PROGRAM MAIN
VAR
	fbSerialCommInstance1 : SerialCom;
	sRecieveString : STRING;
	bRecieveError : BOOL;
	bSendBusy: BOOL;
	eSendError: INT;
	sSendData : STRING;
	bsendTrigger: BOOL;
	STxBuffer: INT;
	tSendTime: INT;
	sizeoff : UINT;
	bRecieveReset: BOOL;
END_VAR

(* Send & Recieve String Data *)
fbSerialCommInstance1(bSendData:= bsendTrigger,
					  bReset := bRecieveReset,
					  TxBuffer := SerialComm.TxBufferPcCom,
					  sSendPrefix:='$01',
					  sSendSuffix:='$02',
					  sSendString:=sSendData,
					  bSendBusy =>bSendBusy,
					  eSendError =>eSendError,
					  RxBuffer := SerialComm.RxBufferPcCom,
					  sReceiveString =>sRecieveString,
					  sReceivePrefix:='$01',
					  sReceiveSuffix:='$02',
					  tReceiveTimeOut := T#1S,
					  bReset :=bRecieveError,
					  bReceiveStringData =>,
					  bReceiveBusy =>,
					  eReceiveError =>,
					  bReceiveTimeOut =>
					  );

END_PROGRAM

(* stored: Version 1.1.0.1, ProductVersion 3.1.4024.11
   POU MAIN: Id {41fc15ba-a291-4be3-a8ad-a005952d4c01}, SpecialFunc None *)
